(* Logix 5000 project; controller PBS_Perfusion vendor 1 type 14 code 217 rev 32.14; software revision 32.03; part 15 of 27 *)
(* tags used below, declared in another part *)
   Inp_Sim : BOOL;   // 1=Simulate working device; 0=Turn ON/OFF actual device
   Cfg_HasPulse : BOOL;   // 1=Enable pulsing functions, 0=On/Off only
   Cfg_CompletePulse : BOOL;   // 1=Finish Pulse when commanded ON or OFF; 0=switch immediately
   Cfg_OperOffPrio : BOOL;   // 1=OCmd_Off any time, 0=OCmd_Off only when Oper selected
   Cfg_OCmdResets : BOOL;   // 1=New device OCmd resets shed latches and cleared alarms, 0=OCmdReset req'd.
   Out : BOOL;   // Primary Output 1=ON, 0=OFF
   Out_Horn : BOOL;   // 1=Sound audible prior to commanded energize/ state change
   Val_Cmd : DINT;   // Device Command: 0=None, 1=Off, 2=On, 3=Pulse Off, 4=Pulse On, 5=Pulse Cont
   Val_Sts : DINT;   // Device Status 0=off 1=on 2=pulse off 3=pulse on 4=pulse cont. 5=turning off 6=turning on
   Val_State : DINT;   // Internal Logic State (for animating STD on faceplate), see manual
   Sts_Out : BOOL;   // 1=Output is ON (energized), 0=Output is OFF (de-energized)
   Sts_Pulsing : BOOL;   // 1=Output is in a pusling sequence
   Sts_Horn : BOOL;   // 1=Horn Active
   Sts_NotRdy : BOOL;   // 1=Device Not Ready, see detail bits for reason
   Sts_Hand : ALIAS FOR CmdSrc.Sts_Hand;
   Sts_Maint : ALIAS FOR CmdSrc.Sts_Maint;
   Sts_Oper : ALIAS FOR CmdSrc.Sts_Oper;
   P_DOut : BOOL;   // Unique Parameter Name for auto - discovery
   Wrk_OffT : TIMER;   // Off Feedback Check Timer
   Wrk_OnT : TIMER;   // On Feedback Check Timer
   Wrk_SimOffT : TIMER;   // Simulation Delay until OFF
   Wrk_SimOnT : TIMER;   // Simulation Delay until ON
   Wrk_OnPulseT : TIMER;   // Output ON Pulse Timer
   Wrk_OffPulseT : TIMER;   // Output OFF Pulse Timer
   Wrk_OffDelayT : TIMER;   // Dealy before turning output OFF (Timer)
   Wrk_OnDelayT : TIMER;   // Delay before turning output ON (Timer)
   Wrk_PermOK : BOOL;   // 1=Permissives are all OK to energize
   Wrk_Cmd : DINT;   // Device Command: 0= None, bit .0=Off, bit .1=On, bit .2=Pulse Off, bit .3=Pulse On, bit .4=Pulse Cont.
   Wrk_NotRdy : BOOL;   // Device Not Ready conditions excluding shed latches
   ORdy_ContPulse : BOOL;   // 1=Ready for OCmd_ContPulse (enables HMI button)
   ORdy_OffPulse : BOOL;   // 1=Ready for OCmd_OffPulse (enables HMI button)
   ORdy_OnPulse : BOOL;   // 1=Ready for OCmd_OnPulse (enables HMI button)
   ORdy_Off : BOOL;   // 1=Ready for OCmd_Off (enables HMI button)
   ORdy_On : BOOL;   // 1=Ready for OCmd_On (enables HMI button)
   Wrk_State : DINT;   // Internal value of state machine current state
   Wrk_StartHorn : BOOL;   // 1=Sound audible prior to commanded energize/ state change
(* P_DOut, continued *)

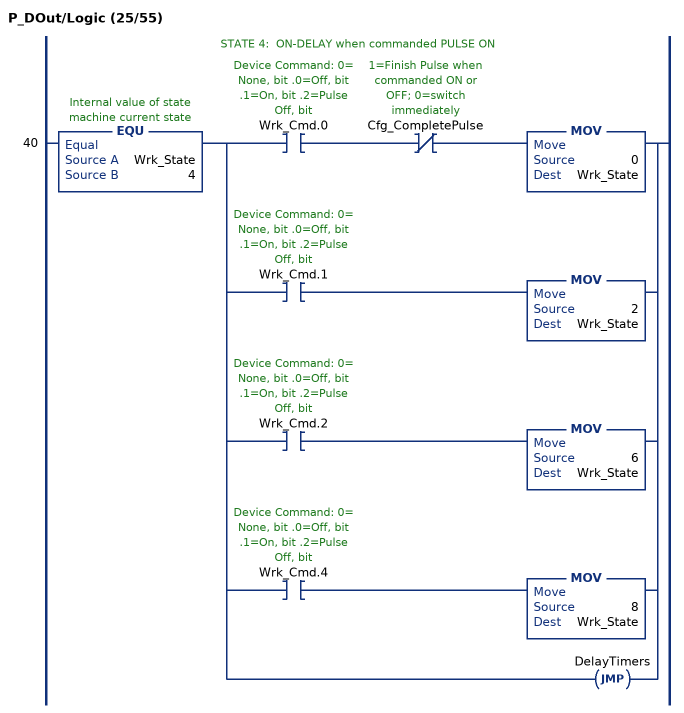
   // STATE 4:  ON-DELAY when commanded PULSE ON
   40: EQU(Wrk_State,4)[XIC(Wrk_Cmd.0) XIO(Cfg_CompletePulse) MOV(0,Wrk_State) ,XIC(Wrk_Cmd.1) MOV(2,Wrk_State) ,XIC(Wrk_Cmd.2) MOV(6,Wrk_State) ,XIC(Wrk_Cmd.4) MOV(8,Wrk_State) ,JMP(DelayTimers) ];
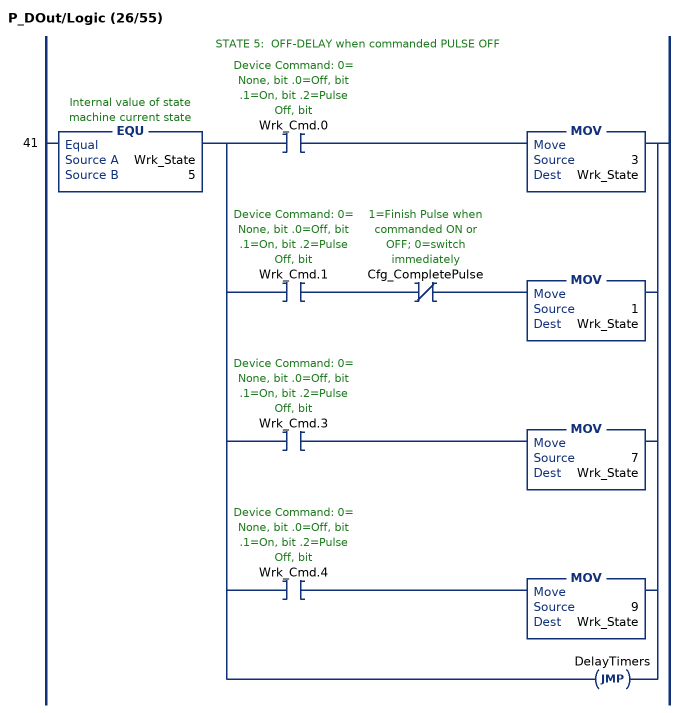
   // STATE 5:  OFF-DELAY when commanded PULSE OFF
   41: EQU(Wrk_State,5)[XIC(Wrk_Cmd.0) MOV(3,Wrk_State) ,XIC(Wrk_Cmd.1) XIO(Cfg_CompletePulse) MOV(1,Wrk_State) ,XIC(Wrk_Cmd.3) MOV(7,Wrk_State) ,XIC(Wrk_Cmd.4) MOV(9,Wrk_State) ,JMP(DelayTimers) ];
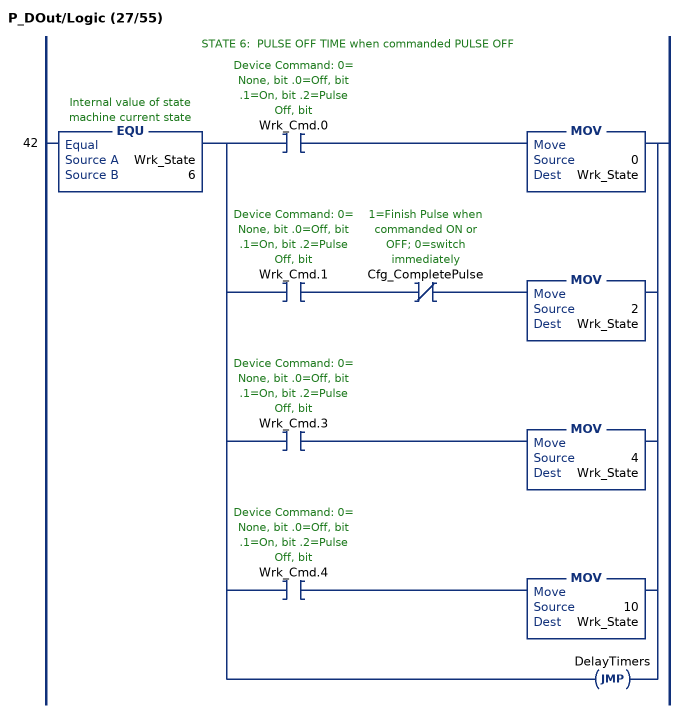
   // STATE 6:  PULSE OFF TIME when commanded PULSE OFF
   42: EQU(Wrk_State,6)[XIC(Wrk_Cmd.0) MOV(0,Wrk_State) ,XIC(Wrk_Cmd.1) XIO(Cfg_CompletePulse) MOV(2,Wrk_State) ,XIC(Wrk_Cmd.3) MOV(4,Wrk_State) ,XIC(Wrk_Cmd.4) MOV(10,Wrk_State) ,JMP(DelayTimers) ];
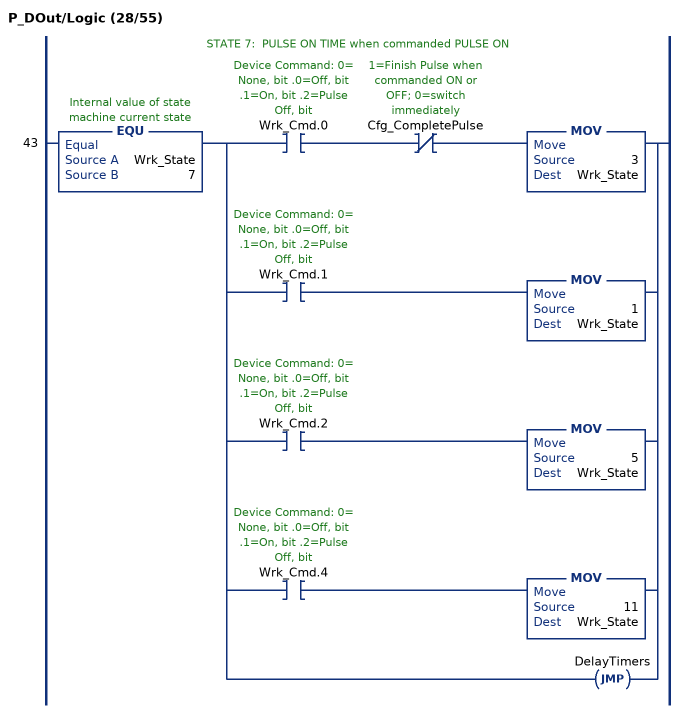
   // STATE 7:  PULSE ON TIME when commanded PULSE ON
   43: EQU(Wrk_State,7)[XIC(Wrk_Cmd.0) XIO(Cfg_CompletePulse) MOV(3,Wrk_State) ,XIC(Wrk_Cmd.1) MOV(1,Wrk_State) ,XIC(Wrk_Cmd.2) MOV(5,Wrk_State) ,XIC(Wrk_Cmd.4) MOV(11,Wrk_State) ,JMP(DelayTimers) ];
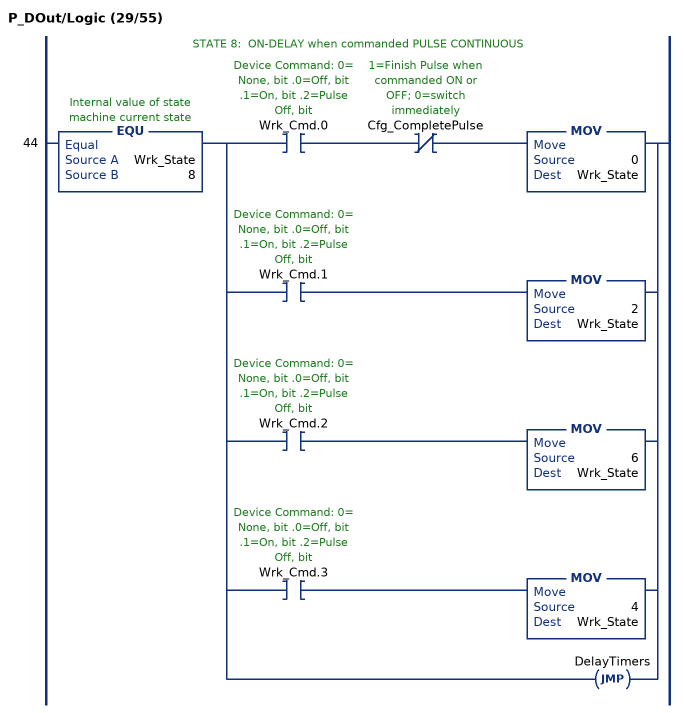
   // STATE 8:  ON-DELAY when commanded PULSE CONTINUOUS
   44: EQU(Wrk_State,8)[XIC(Wrk_Cmd.0) XIO(Cfg_CompletePulse) MOV(0,Wrk_State) ,XIC(Wrk_Cmd.1) MOV(2,Wrk_State) ,XIC(Wrk_Cmd.2) MOV(6,Wrk_State) ,XIC(Wrk_Cmd.3) MOV(4,Wrk_State) ,JMP(DelayTimers) ];
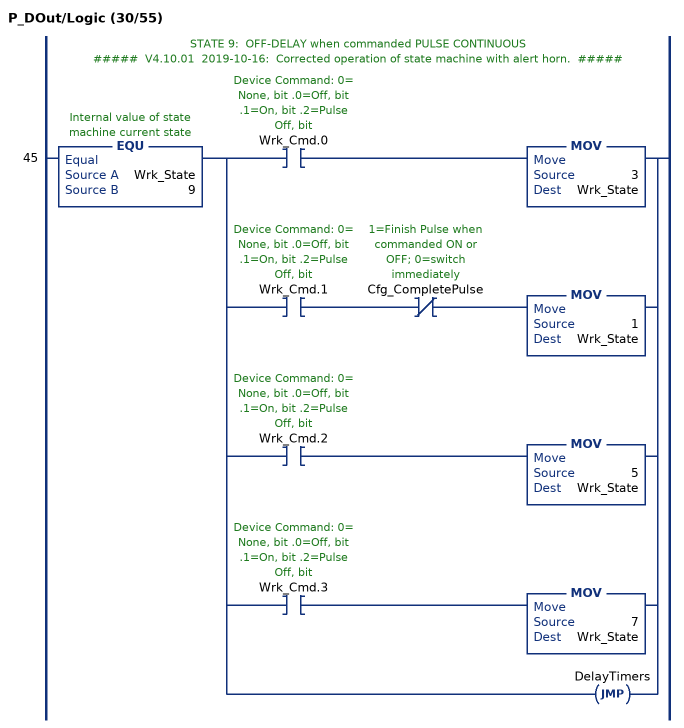
   // STATE 9:  OFF-DELAY when commanded PULSE CONTINUOUS
   // #####  V4.10.01  2019-10-16:  Corrected operation of state machine with alert horn.  #####
   45: EQU(Wrk_State,9)[XIC(Wrk_Cmd.0) MOV(3,Wrk_State) ,XIC(Wrk_Cmd.1) XIO(Cfg_CompletePulse) MOV(1,Wrk_State) ,XIC(Wrk_Cmd.2) MOV(5,Wrk_State) ,XIC(Wrk_Cmd.3) MOV(7,Wrk_State) ,JMP(DelayTimers) ];
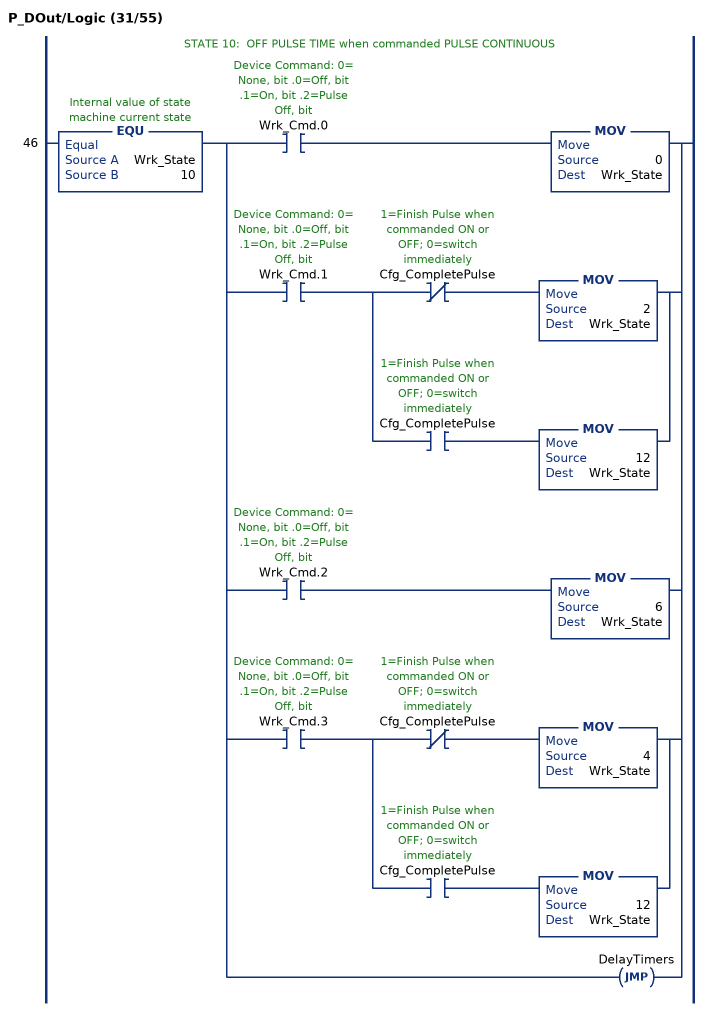
   // STATE 10:  OFF PULSE TIME when commanded PULSE CONTINUOUS
   46: EQU(Wrk_State,10)[XIC(Wrk_Cmd.0) MOV(0,Wrk_State) ,XIC(Wrk_Cmd.1) [XIO(Cfg_CompletePulse) MOV(2,Wrk_State) ,XIC(Cfg_CompletePulse) MOV(12,Wrk_State) ] ,XIC(Wrk_Cmd.2) MOV(6,Wrk_State) ,XIC(Wrk_Cmd.3) [XIO(Cfg_CompletePulse) MOV(4,Wrk_State) ,XIC(Cfg_CompletePulse) MOV(12,Wrk_State) ] ,JMP(DelayTimers) ];
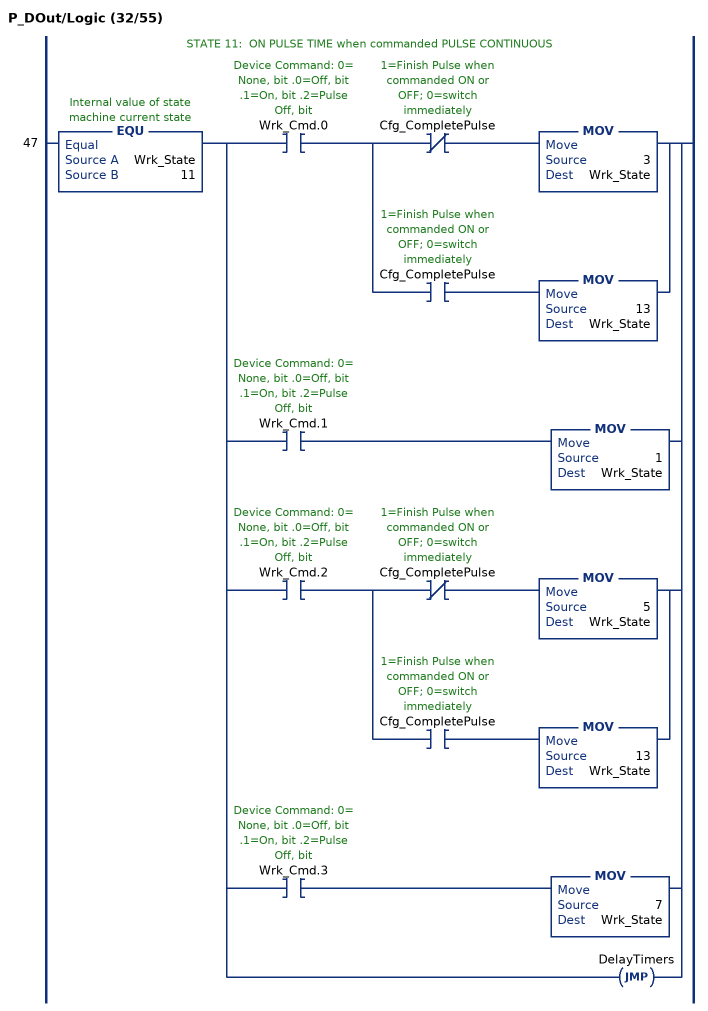
   // STATE 11:  ON PULSE TIME when commanded PULSE CONTINUOUS
   47: EQU(Wrk_State,11)[XIC(Wrk_Cmd.0) [XIO(Cfg_CompletePulse) MOV(3,Wrk_State) ,XIC(Cfg_CompletePulse) MOV(13,Wrk_State) ] ,XIC(Wrk_Cmd.1) MOV(1,Wrk_State) ,XIC(Wrk_Cmd.2) [XIO(Cfg_CompletePulse) MOV(5,Wrk_State) ,XIC(Cfg_CompletePulse) MOV(13,Wrk_State) ] ,XIC(Wrk_Cmd.3) MOV(7,Wrk_State) ,JMP(DelayTimers) ];
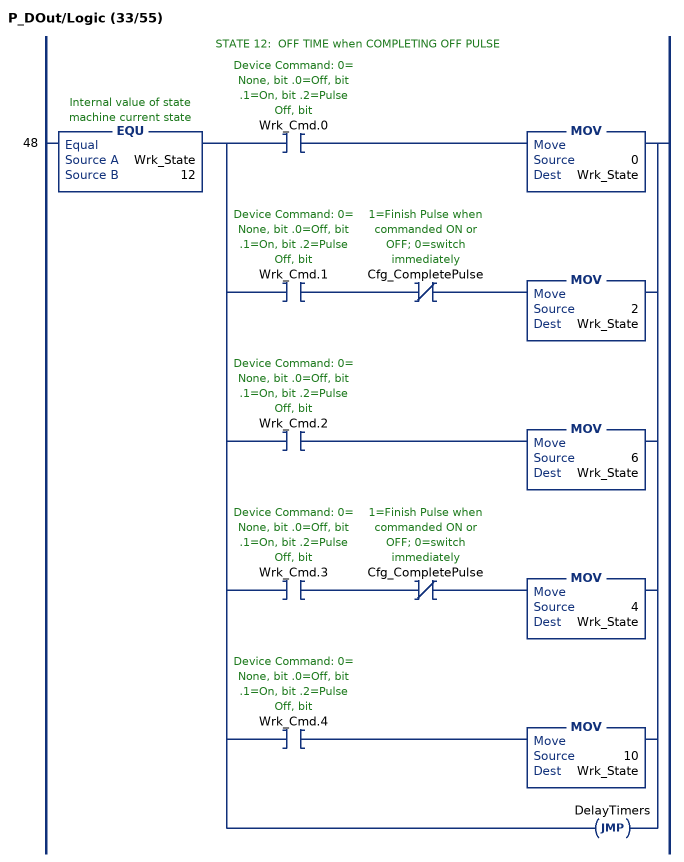
   // STATE 12:  OFF TIME when COMPLETING OFF PULSE
   48: EQU(Wrk_State,12)[XIC(Wrk_Cmd.0) MOV(0,Wrk_State) ,XIC(Wrk_Cmd.1) XIO(Cfg_CompletePulse) MOV(2,Wrk_State) ,XIC(Wrk_Cmd.2) MOV(6,Wrk_State) ,XIC(Wrk_Cmd.3) XIO(Cfg_CompletePulse) MOV(4,Wrk_State) ,XIC(Wrk_Cmd.4) MOV(10,Wrk_State) ,JMP(DelayTimers) ];
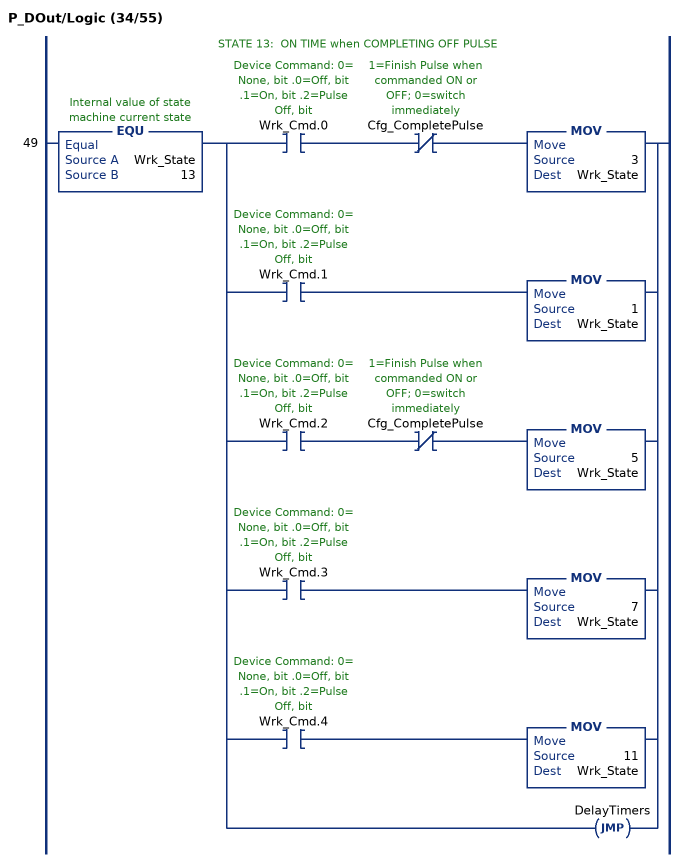
   // STATE 13:  ON TIME when COMPLETING OFF PULSE
   49: EQU(Wrk_State,13)[XIC(Wrk_Cmd.0) XIO(Cfg_CompletePulse) MOV(3,Wrk_State) ,XIC(Wrk_Cmd.1) MOV(1,Wrk_State) ,XIC(Wrk_Cmd.2) XIO(Cfg_CompletePulse) MOV(5,Wrk_State) ,XIC(Wrk_Cmd.3) MOV(7,Wrk_State) ,XIC(Wrk_Cmd.4) MOV(11,Wrk_State) ,JMP(DelayTimers) ];
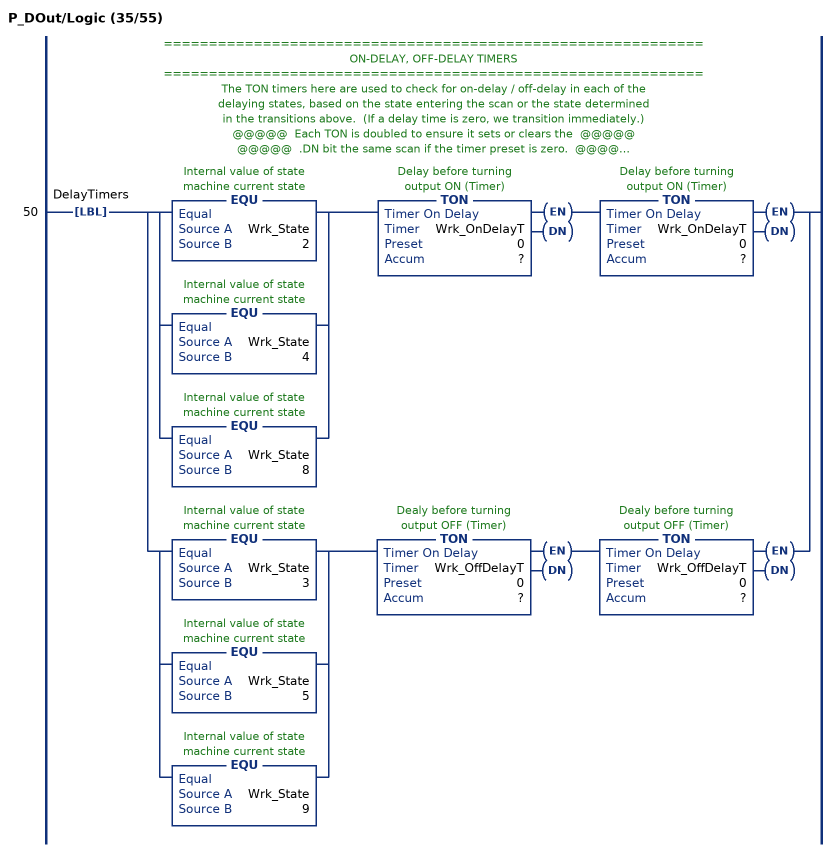
   // ============================================================
   // ON-DELAY, OFF-DELAY TIMERS
   // ============================================================
   // The TON timers here are used to check for on-delay / off-delay in each of the
   // delaying states, based on the state entering the scan or the state determined
   // in the transitions above.  (If a delay time is zero, we transition immediately.)
   // @@@@@  Each TON is doubled to ensure it sets or clears the  @@@@@
   // @@@@@  .DN bit the same scan if the timer preset is zero.  @@@@@
   // The Timers will be disabled while Horn is active, preventing change of state
   // #####  V4.10.00  2019-03-08:  Added audible alert on commanded energize/state change.  #####
   // #####  V4.10.01  2019-10-16:  Corrected operation of state machine with alert horn.  #####
   50: LBL(DelayTimers)[[EQU(Wrk_State,2) ,EQU(Wrk_State,4) ,EQU(Wrk_State,8) ] TON(Wrk_OnDelayT,?,?) TON(Wrk_OnDelayT,?,?) ,[EQU(Wrk_State,3) ,EQU(Wrk_State,5) ,EQU(Wrk_State,9) ] TON(Wrk_OffDelayT,?,?) TON(Wrk_OffDelayT,?,?) ];
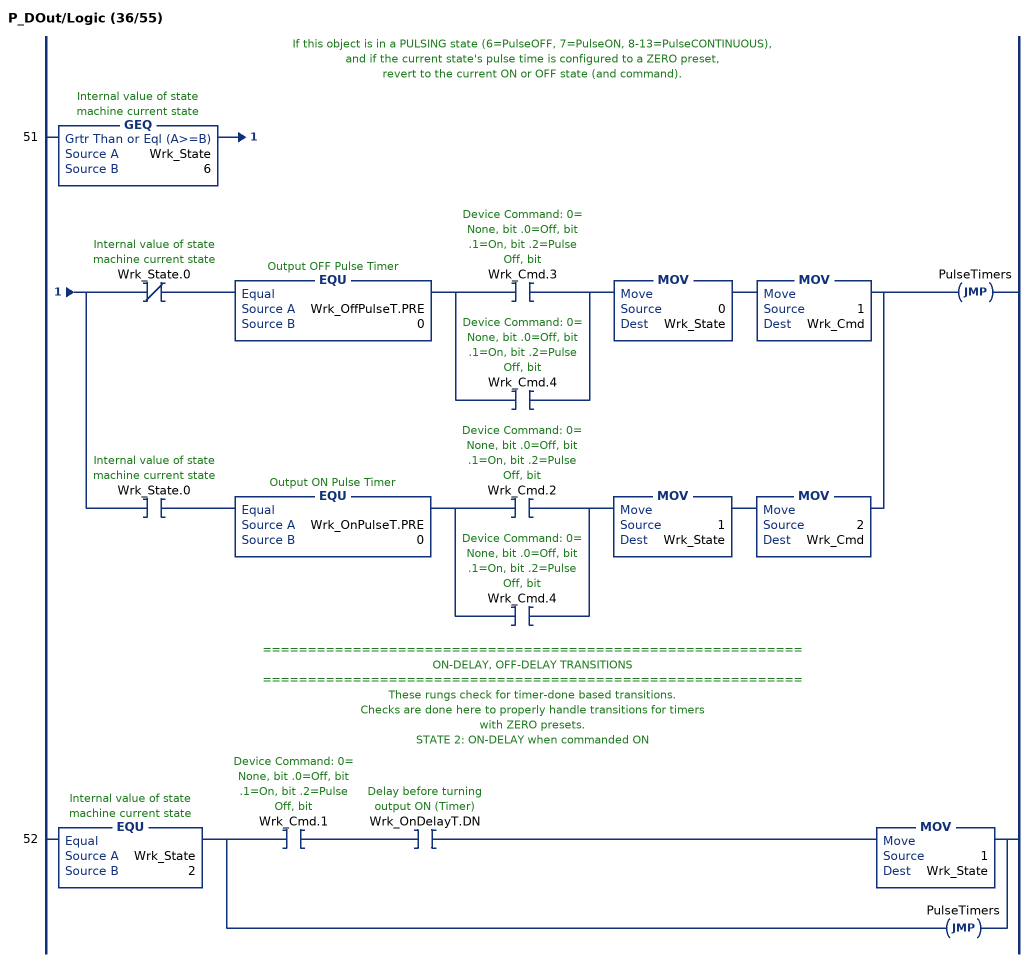
   // If this object is in a PULSING state (6=PulseOFF, 7=PulseON, 8-13=PulseCONTINUOUS),
   // and if the current state's pulse time is configured to a ZERO preset,
   // revert to the current ON or OFF state (and command).
   51: GEQ(Wrk_State,6)[XIO(Wrk_State.0) EQU(Wrk_OffPulseT.PRE,0) [XIC(Wrk_Cmd.3) ,XIC(Wrk_Cmd.4) ] MOV(0,Wrk_State) MOV(1,Wrk_Cmd) ,XIC(Wrk_State.0) EQU(Wrk_OnPulseT.PRE,0) [XIC(Wrk_Cmd.2) ,XIC(Wrk_Cmd.4) ] MOV(1,Wrk_State) MOV(2,Wrk_Cmd) ]JMP(PulseTimers);
   // ============================================================
   // ON-DELAY, OFF-DELAY TRANSITIONS
   // ============================================================
   // These rungs check for timer-done based transitions.
   // Checks are done here to properly handle transitions for timers
   // with ZERO presets.
   // STATE 2: ON-DELAY when commanded ON
   52: EQU(Wrk_State,2)[XIC(Wrk_Cmd.1) XIC(Wrk_OnDelayT.DN) MOV(1,Wrk_State) ,JMP(PulseTimers) ];
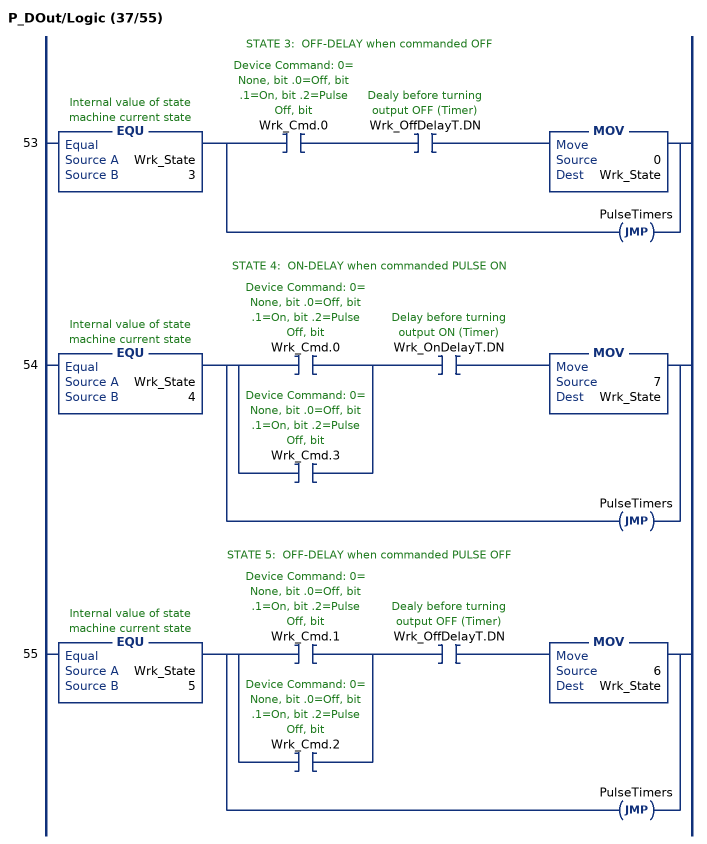
   // STATE 3:  OFF-DELAY when commanded OFF
   53: EQU(Wrk_State,3)[XIC(Wrk_Cmd.0) XIC(Wrk_OffDelayT.DN) MOV(0,Wrk_State) ,JMP(PulseTimers) ];
   // STATE 4:  ON-DELAY when commanded PULSE ON
   54: EQU(Wrk_State,4)[[XIC(Wrk_Cmd.0) ,XIC(Wrk_Cmd.3) ] XIC(Wrk_OnDelayT.DN) MOV(7,Wrk_State) ,JMP(PulseTimers) ];
   // STATE 5:  OFF-DELAY when commanded PULSE OFF
   55: EQU(Wrk_State,5)[[XIC(Wrk_Cmd.1) ,XIC(Wrk_Cmd.2) ] XIC(Wrk_OffDelayT.DN) MOV(6,Wrk_State) ,JMP(PulseTimers) ];
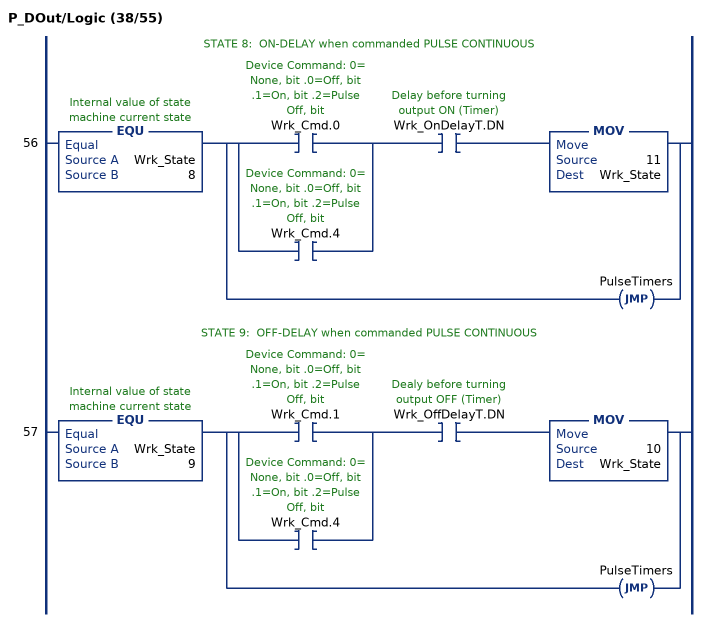
   // STATE 8:  ON-DELAY when commanded PULSE CONTINUOUS
   56: EQU(Wrk_State,8)[[XIC(Wrk_Cmd.0) ,XIC(Wrk_Cmd.4) ] XIC(Wrk_OnDelayT.DN) MOV(11,Wrk_State) ,JMP(PulseTimers) ];
   // STATE 9:  OFF-DELAY when commanded PULSE CONTINUOUS
   57: EQU(Wrk_State,9)[[XIC(Wrk_Cmd.1) ,XIC(Wrk_Cmd.4) ] XIC(Wrk_OffDelayT.DN) MOV(10,Wrk_State) ,JMP(PulseTimers) ];
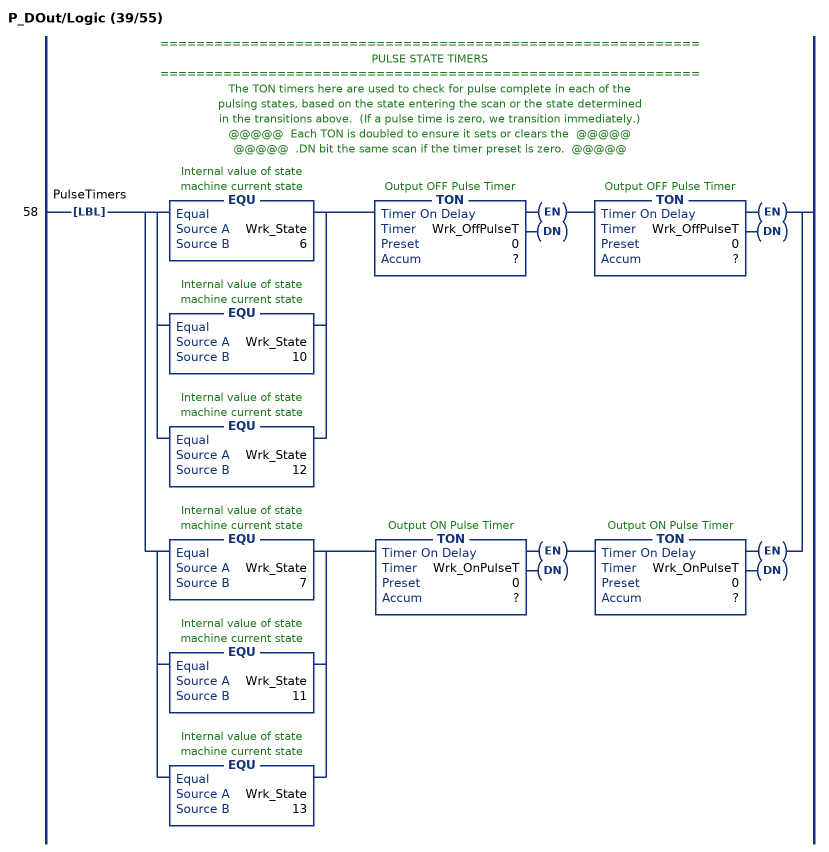
   // ============================================================
   // PULSE STATE TIMERS
   // ============================================================
   // The TON timers here are used to check for pulse complete in each of the
   // pulsing states, based on the state entering the scan or the state determined
   // in the transitions above.  (If a pulse time is zero, we transition immediately.)
   // @@@@@  Each TON is doubled to ensure it sets or clears the  @@@@@
   // @@@@@  .DN bit the same scan if the timer preset is zero.  @@@@@
   58: LBL(PulseTimers)[[EQU(Wrk_State,6) ,EQU(Wrk_State,10) ,EQU(Wrk_State,12) ] TON(Wrk_OffPulseT,?,?) TON(Wrk_OffPulseT,?,?) ,[EQU(Wrk_State,7) ,EQU(Wrk_State,11) ,EQU(Wrk_State,13) ] TON(Wrk_OnPulseT,?,?) TON(Wrk_OnPulseT,?,?) ];
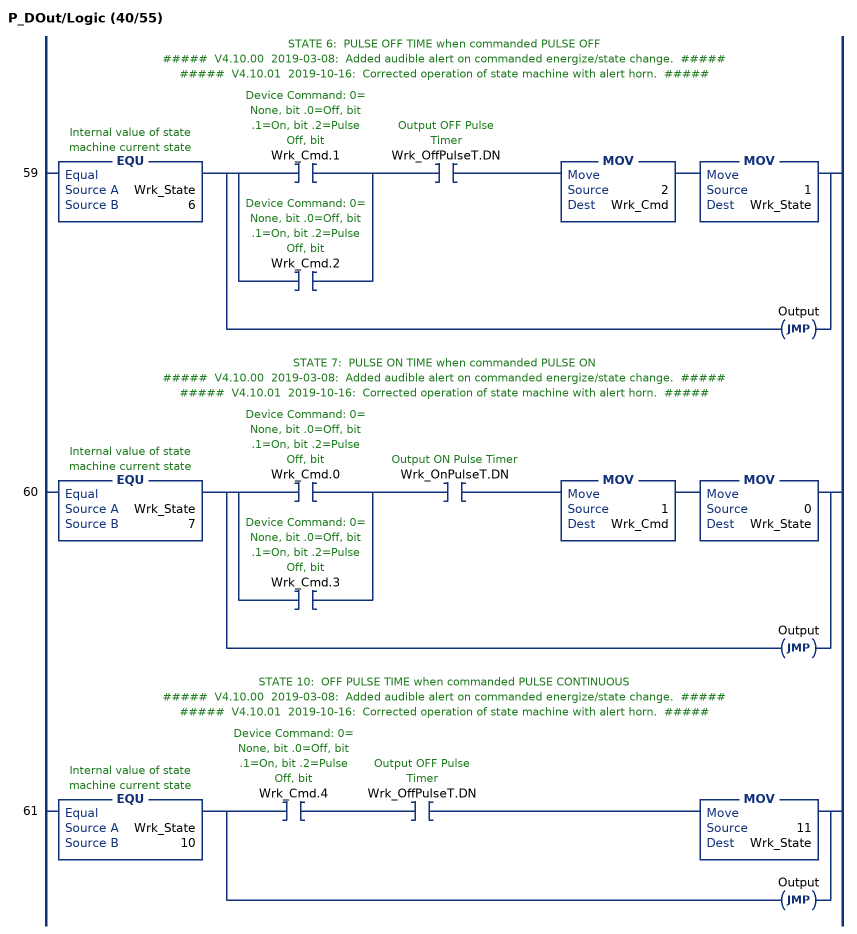
   // STATE 6:  PULSE OFF TIME when commanded PULSE OFF
   // #####  V4.10.00  2019-03-08:  Added audible alert on commanded energize/state change.  #####
   // #####  V4.10.01  2019-10-16:  Corrected operation of state machine with alert horn.  #####
   59: EQU(Wrk_State,6)[[XIC(Wrk_Cmd.1) ,XIC(Wrk_Cmd.2) ] XIC(Wrk_OffPulseT.DN) MOV(2,Wrk_Cmd) MOV(1,Wrk_State) ,JMP(Output) ];
   // STATE 7:  PULSE ON TIME when commanded PULSE ON
   // #####  V4.10.00  2019-03-08:  Added audible alert on commanded energize/state change.  #####
   // #####  V4.10.01  2019-10-16:  Corrected operation of state machine with alert horn.  #####
   60: EQU(Wrk_State,7)[[XIC(Wrk_Cmd.0) ,XIC(Wrk_Cmd.3) ] XIC(Wrk_OnPulseT.DN) MOV(1,Wrk_Cmd) MOV(0,Wrk_State) ,JMP(Output) ];
   // STATE 10:  OFF PULSE TIME when commanded PULSE CONTINUOUS
   // #####  V4.10.00  2019-03-08:  Added audible alert on commanded energize/state change.  #####
   // #####  V4.10.01  2019-10-16:  Corrected operation of state machine with alert horn.  #####
   61: EQU(Wrk_State,10)[XIC(Wrk_Cmd.4) XIC(Wrk_OffPulseT.DN) MOV(11,Wrk_State) ,JMP(Output) ];
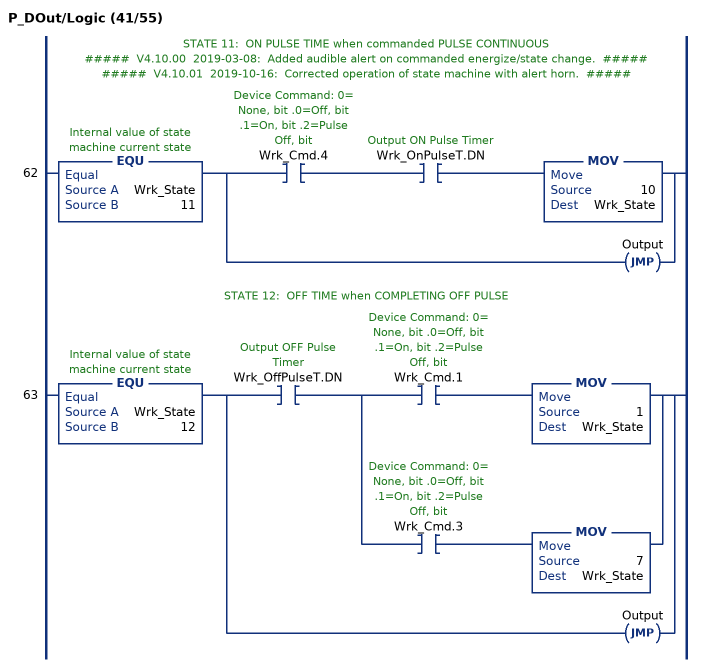
   // STATE 11:  ON PULSE TIME when commanded PULSE CONTINUOUS
   // #####  V4.10.00  2019-03-08:  Added audible alert on commanded energize/state change.  #####
   // #####  V4.10.01  2019-10-16:  Corrected operation of state machine with alert horn.  #####
   62: EQU(Wrk_State,11)[XIC(Wrk_Cmd.4) XIC(Wrk_OnPulseT.DN) MOV(10,Wrk_State) ,JMP(Output) ];
   // STATE 12:  OFF TIME when COMPLETING OFF PULSE
   63: EQU(Wrk_State,12)[XIC(Wrk_OffPulseT.DN) [XIC(Wrk_Cmd.1) MOV(1,Wrk_State) ,XIC(Wrk_Cmd.3) MOV(7,Wrk_State) ] ,JMP(Output) ];
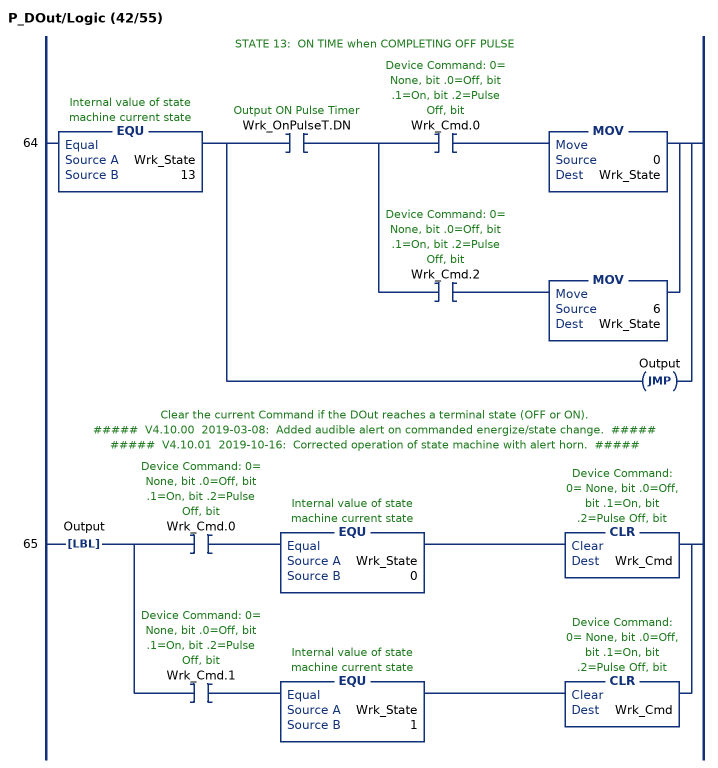
   // STATE 13:  ON TIME when COMPLETING OFF PULSE
   64: EQU(Wrk_State,13)[XIC(Wrk_OnPulseT.DN) [XIC(Wrk_Cmd.0) MOV(0,Wrk_State) ,XIC(Wrk_Cmd.2) MOV(6,Wrk_State) ] ,JMP(Output) ];
   // Clear the current Command if the DOut reaches a terminal state (OFF or ON).
   // #####  V4.10.00  2019-03-08:  Added audible alert on commanded energize/state change.  #####
   // #####  V4.10.01  2019-10-16:  Corrected operation of state machine with alert horn.  #####
   65: LBL(Output)[XIC(Wrk_Cmd.0) EQU(Wrk_State,0) CLR(Wrk_Cmd) ,XIC(Wrk_Cmd.1) EQU(Wrk_State,1) CLR(Wrk_Cmd) ];
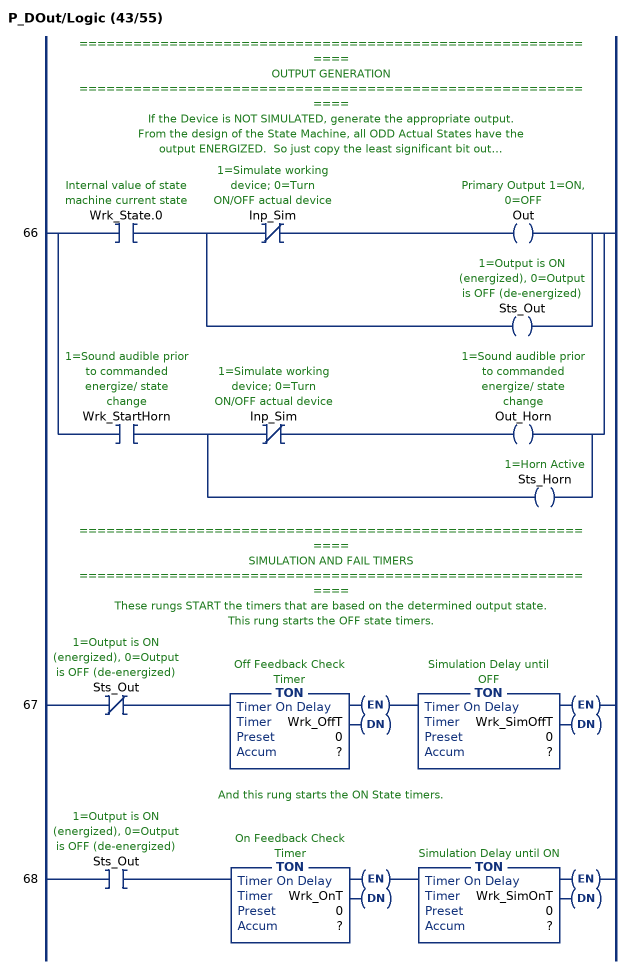
   // ============================================================
   // OUTPUT GENERATION
   // ============================================================
   // If the Device is NOT SIMULATED, generate the appropriate output.
   // From the design of the State Machine, all ODD Actual States have the
   // output ENERGIZED.  So just copy the least significant bit out!
   // #####  V4.10.00  2019-03-08:  Added audible alert on commanded energize/state change.  #####
   66: [XIC(Wrk_State.0) [XIO(Inp_Sim) OTE(Out) ,OTE(Sts_Out) ] ,XIC(Wrk_StartHorn) [XIO(Inp_Sim) OTE(Out_Horn) ,OTE(Sts_Horn) ] ];
   // ============================================================
   // SIMULATION AND FAIL TIMERS
   // ============================================================
   // These rungs START the timers that are based on the determined output state.
   // This rung starts the OFF state timers.
   67: XIO(Sts_Out)TON(Wrk_OffT,?,?)TON(Wrk_SimOffT,?,?);
   // And this rung starts the ON State timers.
   68: XIC(Sts_Out)TON(Wrk_OnT,?,?)TON(Wrk_SimOnT,?,?);
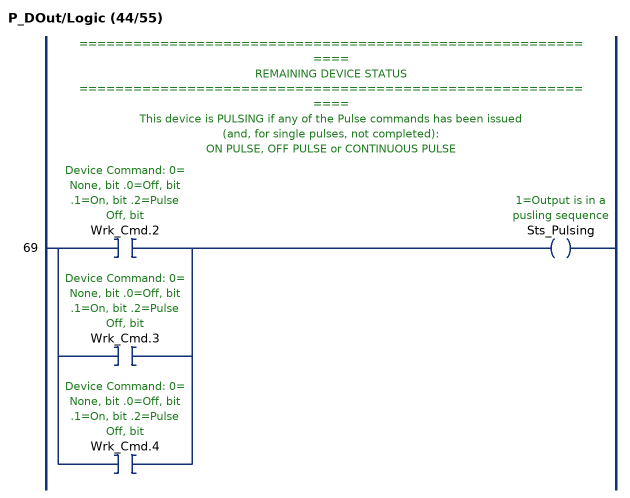
   // ============================================================
   // REMAINING DEVICE STATUS
   // ============================================================
   // This device is PULSING if any of the Pulse commands has been issued
   // (and, for single pulses, not completed):
   // ON PULSE, OFF PULSE or CONTINUOUS PULSE
   69: [XIC(Wrk_Cmd.2) ,XIC(Wrk_Cmd.3) ,XIC(Wrk_Cmd.4) ]OTE(Sts_Pulsing);
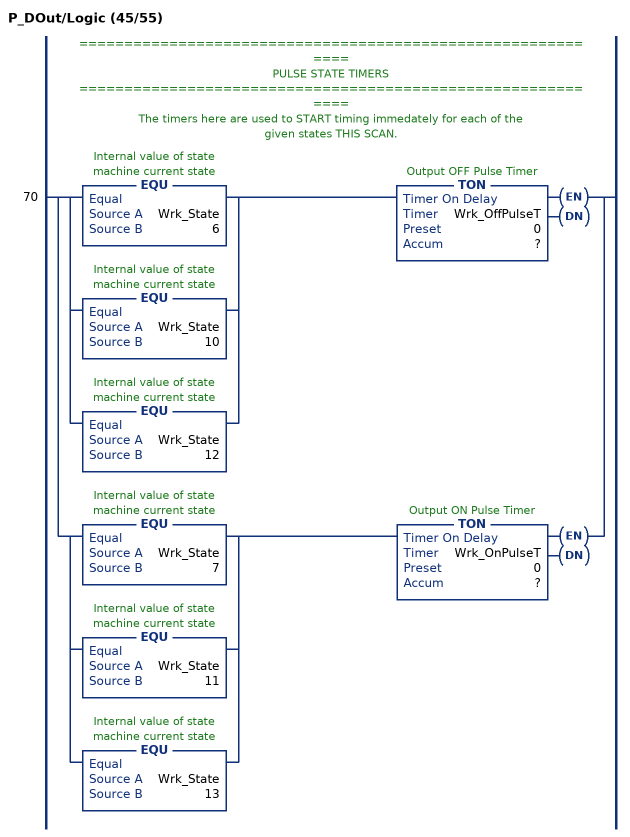
   // ============================================================
   // PULSE STATE TIMERS
   // ============================================================
   // The timers here are used to START timing immedately for each of the
   // given states THIS SCAN.
   70: [[EQU(Wrk_State,6) ,EQU(Wrk_State,10) ,EQU(Wrk_State,12) ] TON(Wrk_OffPulseT,?,?) ,[EQU(Wrk_State,7) ,EQU(Wrk_State,11) ,EQU(Wrk_State,13) ] TON(Wrk_OnPulseT,?,?) ];
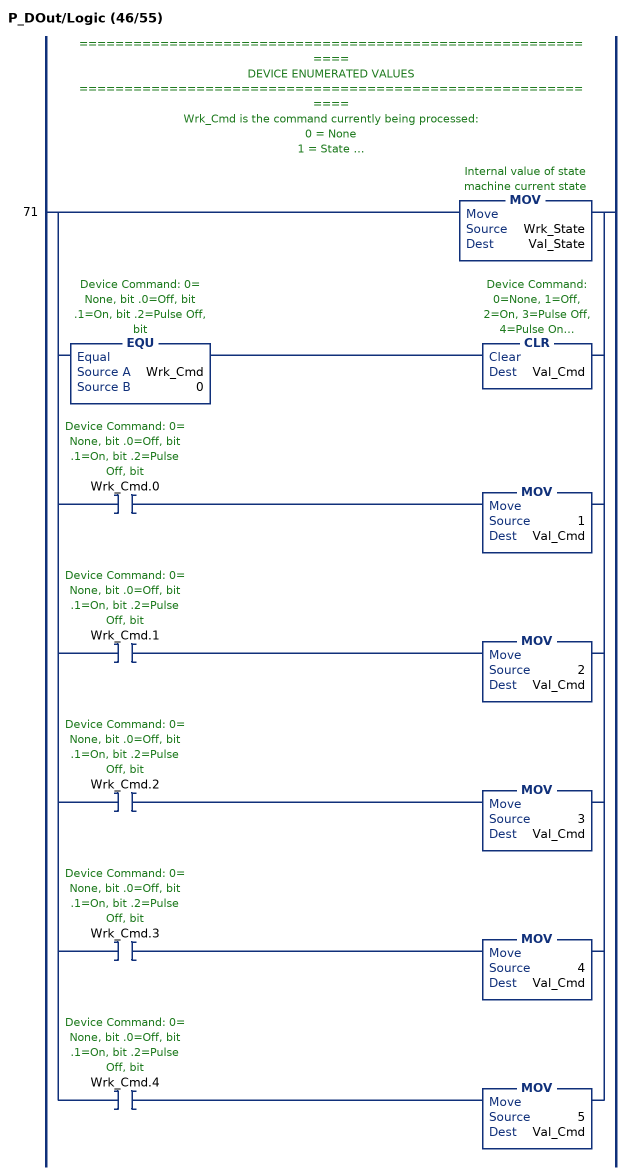
   // ============================================================
   // DEVICE ENUMERATED VALUES
   // ============================================================
   // Wrk_Cmd is the command currently being processed:
   // 0 = None
   // 1 = State 0
   // 2 = State 1
   // 3 = State 2
   // 4 = State 3
   // Wrk_State is the internal state machine state:
   // 0 = OFF
   // 1 = ON
   // 2 = ON command ON-DELAY
   // 3 = OFF command OFF-DELAY
   // 4 = PULSE ON command ON-DELAY
   // 5 = PULSE OFF command OFF-DELAY
   // 6 = PULSE ON command ON PULSE time
   // 7 = PULSE OFF command OFF PULSE time
   // 8 = PULSE CONTINUOUS command ON-DELAY
   // 9 = PULSE CONTINUOUS command OFF-DELAY
   // 10 = PULSE CONTINUOUS command OFF PULSE time
   // 11 = PULSE CONTINUOUS command ON PULSE time
   // 12 = OFF PULSE completion time
   // 13 = ON PULSE completion time
   71: [MOV(Wrk_State,Val_State) ,EQU(Wrk_Cmd,0) CLR(Val_Cmd) ,XIC(Wrk_Cmd.0) MOV(1,Val_Cmd) ,XIC(Wrk_Cmd.1) MOV(2,Val_Cmd) ,XIC(Wrk_Cmd.2) MOV(3,Val_Cmd) ,XIC(Wrk_Cmd.3) MOV(4,Val_Cmd) ,XIC(Wrk_Cmd.4) MOV(5,Val_Cmd) ];
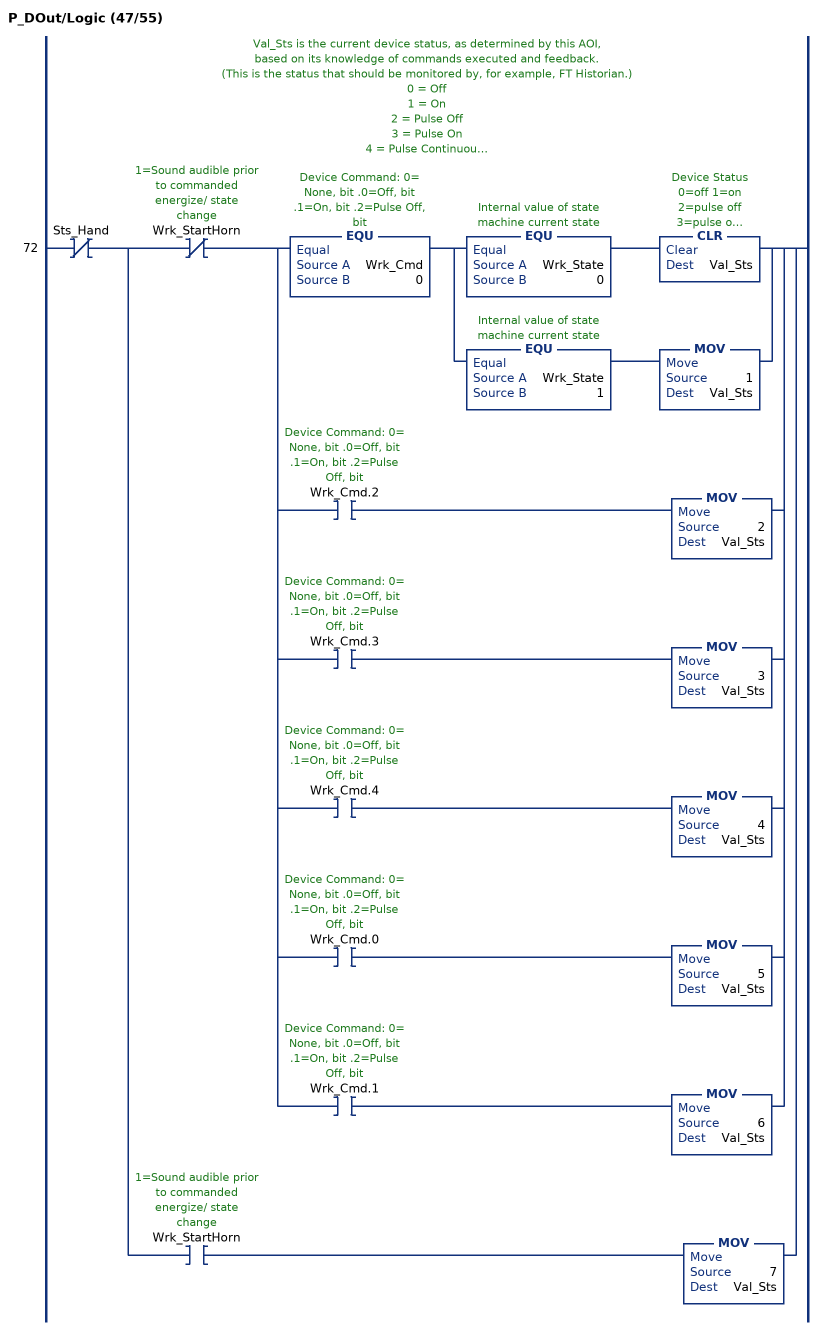
   // Val_Sts is the current device status, as determined by this AOI,
   // based on its knowledge of commands executed and feedback.
   // (This is the status that should be monitored by, for example, FT Historian.)
   // 0 = Off
   // 1 = On
   // 2 = Pulse Off
   // 3 = Pulse On
   // 4 = Pulse Continuous
   // 5 = Turning On
   // 6 = Turning Off
   // 7 = Horn
   // 33 = Out of Service (here or in EnableInFalse routine)
   // #####  V4.00.00  2018-07-02: Using P_CmdSrc, Disabled replaced by Out of Service.  #####
   // #####  V4.10.00  2019-03-08:  Added Horn Status.  #####
   72: XIO(Sts_Hand)[XIO(Wrk_StartHorn) [EQU(Wrk_Cmd,0) [EQU(Wrk_State,0) CLR(Val_Sts) ,EQU(Wrk_State,1) MOV(1,Val_Sts) ] ,XIC(Wrk_Cmd.2) MOV(2,Val_Sts) ,XIC(Wrk_Cmd.3) MOV(3,Val_Sts) ,XIC(Wrk_Cmd.4) MOV(4,Val_Sts) ,XIC(Wrk_Cmd.0) MOV(5,Val_Sts) ,XIC(Wrk_Cmd.1) MOV(6,Val_Sts) ] ,XIC(Wrk_StartHorn) MOV(7,Val_Sts) ];
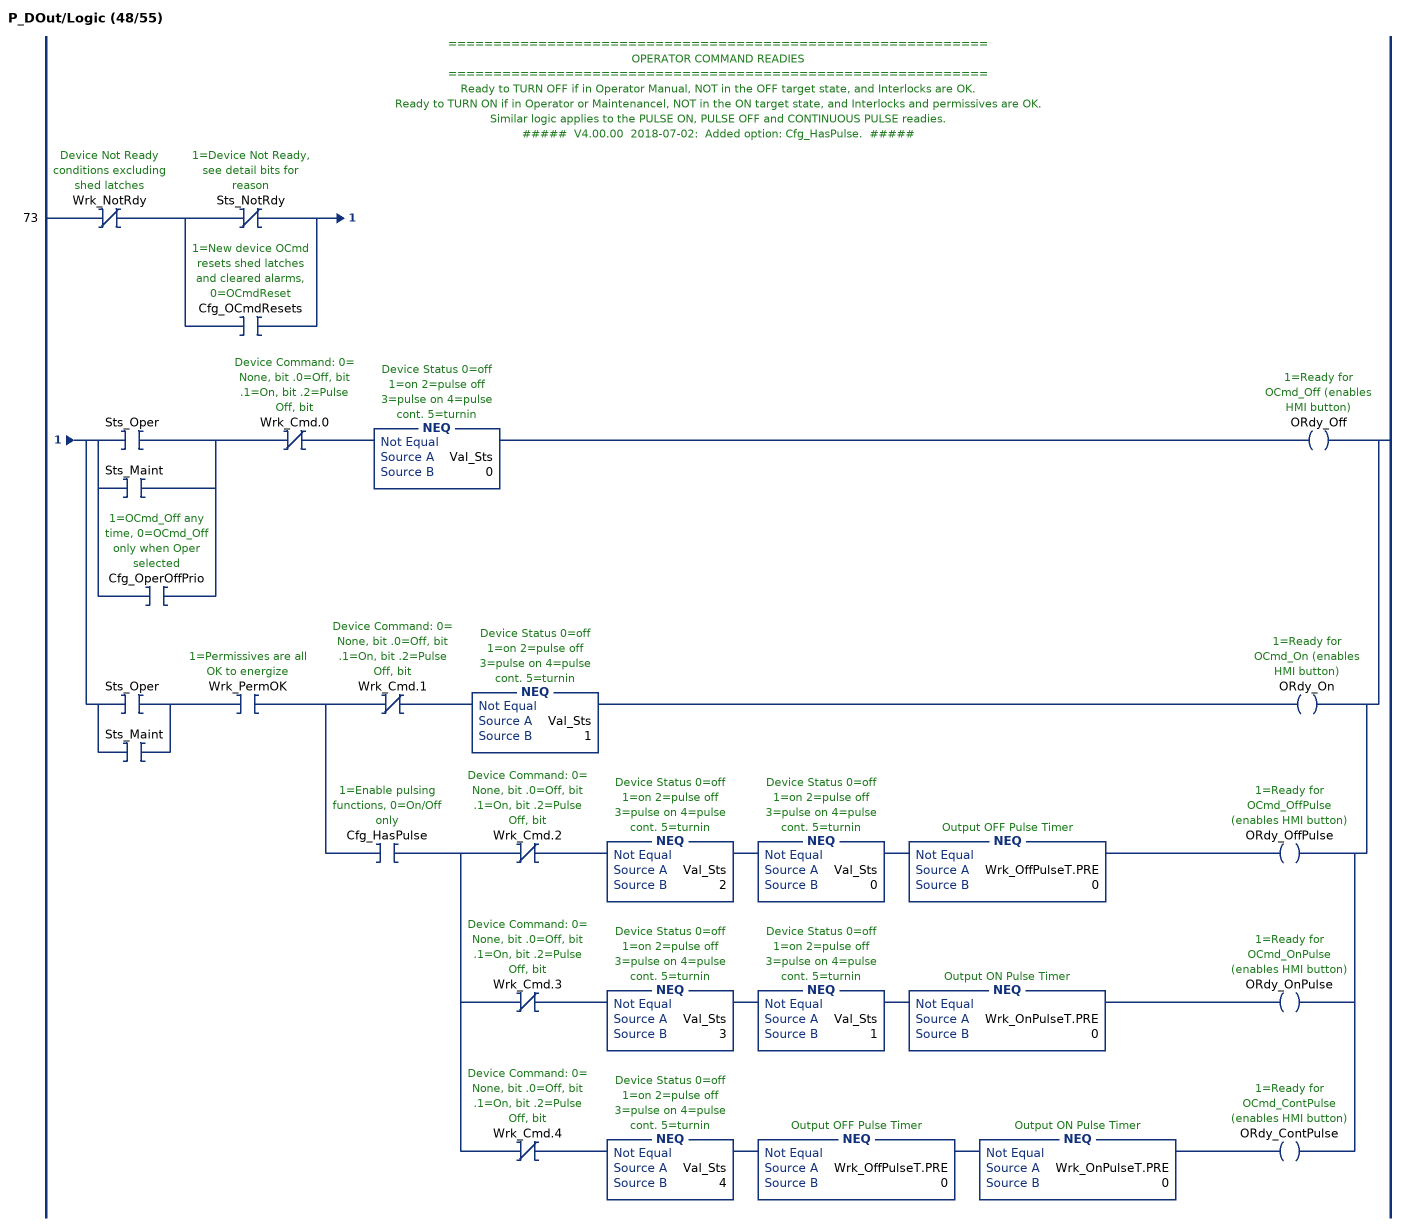
   // ============================================================
   // OPERATOR COMMAND READIES
   // ============================================================
   // Ready to TURN OFF if in Operator Manual, NOT in the OFF target state, and Interlocks are OK.
   // Ready to TURN ON if in Operator or Maintenancel, NOT in the ON target state, and Interlocks and permissives are OK.
   // Similar logic applies to the PULSE ON, PULSE OFF and CONTINUOUS PULSE readies.
   // #####  V4.00.00  2018-07-02:  Added option: Cfg_HasPulse.  #####
   73: XIO(Wrk_NotRdy)[XIO(Sts_NotRdy) ,XIC(Cfg_OCmdResets) ][[XIC(Sts_Oper) ,XIC(Sts_Maint) ,XIC(Cfg_OperOffPrio) ] XIO(Wrk_Cmd.0) NEQ(Val_Sts,0) OTE(ORdy_Off) ,[XIC(Sts_Oper) ,XIC(Sts_Maint) ] XIC(Wrk_PermOK) [XIO(Wrk_Cmd.1) NEQ(Val_Sts,1) OTE(ORdy_On) ,XIC(Cfg_HasPulse) [XIO(Wrk_Cmd.2) NEQ(Val_Sts,2) NEQ(Val_Sts,0) NEQ(Wrk_OffPulseT.PRE,0) OTE(ORdy_OffPulse) ,XIO(Wrk_Cmd.3) NEQ(Val_Sts,3) NEQ(Val_Sts,1) NEQ(Wrk_OnPulseT.PRE,0) OTE(ORdy_OnPulse) ,XIO(Wrk_Cmd.4) NEQ(Val_Sts,4) NEQ(Wrk_OffPulseT.PRE,0) NEQ(Wrk_OnPulseT.PRE,0) OTE(ORdy_ContPulse) ] ] ];
